{attribute 'TcGenerated'}
{attribute 'no-analysis'}
{attribute 'linkalways'}
// This function has been automatically generated from the project information.
VAR_GLOBAL CONSTANT
	{attribute 'const_non_replaced'}
	stLibVersion_ESO_LDC_Timer_Library : ST_LibVersion := (iMajor := 1, iMinor := 0, iBuild := 5, iRevision := 0, nFlags := 0, sVersion := '1.0.5.0');
END_VAR

(* stored: Version 1.1.0.1, ProductVersion 3.1.4024.11
   GVL Global_Version: Id {73bf87b5-3491-4cc9-b29f-d3551a02dc3d} *)
